TYPE UDT_PlcStatus_RD :
STRUCT
  
cycleTime : TIME; // 周期时间
maxCycleTime : Time; // 最长循环时间
minCycleTime : Time; // 最短循环时间
systemClock : DATE_AND_TIME; // 系统时钟
localClock : DATE_AND_TIME; // 本地时钟
status : Int; // CPU运行状态

END_STRUCT
END_TYPE

(* stored: Version 1.1.0.1, ProductVersion 3.1.4024.12
   DUT UDT_PlcStatus_RD: Id {7b780c59-0e2f-4fb1-8235-4c0866bced8a} *)
